(*
SPDX-FileCopyrightText: © 2026 Oleksandr Tiutyk <trofimich@gmail.com>
SPDX-License-Identifier: MIT
License: https://opensource.org/license/mit
*)

(*!
<summary>Defines a boolean predicate evaluated by workflow activities.</summary>
*)

INTERFACE ICondition EXTENDS IWorkflowElement

(*!
<summary>Reports whether the condition is completely configured and ready for evaluation.</summary>
*)
{attribute 'monitoring' := 'call'}
PROPERTY Configured : BOOL
GET
END_GET
END_PROPERTY

(*!
<summary>Evaluates the condition in the context of the specified activity.</summary>
<param name="activity">Activity requesting evaluation, used for variable lookup context.</param>
*)
METHOD Evaluate : BOOL
VAR_INPUT
	activity : IActivity;
END_VAR
END_METHOD

(*!
<summary>Resolves the nearest activity that hosts this condition, traversing parent conditions if needed.</summary>
<description>
Returns the direct ParentActivity when attached directly to an activity, or traverses the ParentCondition
chain upward until the hosting activity is found. Returns 0 if unattached.
</description>
*)
{attribute 'monitoring' := 'call'}
PROPERTY EnclosingActivity : IActivity
GET
END_GET
END_PROPERTY

(*!
<summary>Gets or sets the borrowed immediate parent activity to which this condition is attached.</summary>
<description>
Returns 0 when the condition is attached to a parent condition rather than directly to an activity.
Use EnclosingActivity to resolve the owning activity context through the parent condition chain.
The standard implementation validates cycles, fixed workflow association and PASSIVE_READY before a new
link is stored. Existing parent links cannot be detached or replaced; an unchanged link is a no-op.
Parents are borrowed for the tree lifetime and do not transfer ownership. Configuration is single-task
without reentry; a child with a known owner requires a parent from that same known workflow.
</description>
*)
{attribute 'monitoring' := 'call'}
PROPERTY ParentActivity : IActivity
GET
END_GET
SET
END_SET
END_PROPERTY

(*!
<summary>Gets or sets the borrowed parent composite condition to which this condition is attached.</summary>
<description>
The standard implementation validates cycles, fixed workflow association and PASSIVE_READY before a new
link is stored. Existing parent links cannot be detached or replaced; an unchanged link is a no-op.
Parents are borrowed for the tree lifetime and do not transfer ownership. Configuration is single-task
without reentry; a child with a known owner requires a parent from that same known workflow.
</description>
*)
{attribute 'monitoring' := 'call'}
PROPERTY ParentCondition : ICondition
GET
END_GET
SET
END_SET
END_PROPERTY

END_INTERFACE

(* stored: Version 1.1.0.1
   Itf ICondition: Id {19c0280f-d2f8-424c-8f16-7278f6083af3}
   Property Configured: Id {be75d7d4-64bd-40dc-bf90-f31d9ada671d}
   Get Get: Id {2cba87ee-59ce-4e78-adf7-b7ddc27d2a6b}
   Method Evaluate: Id {10c78263-1c71-45c9-9b13-37be129d2d1c}
   Property EnclosingActivity: Id {bafd7227-41ac-4f1b-8902-4752d6ce1cbf}
   Get Get: Id {36cff938-a908-479f-9391-58af2b4987b2}
   Property ParentActivity: Id {336055e4-538d-4d26-b32a-4579c4dcea29}
   Get Get: Id {ee7ae3cd-f785-417e-8de6-667289c8af2c}
   Set Set: Id {5479ead8-c01c-4380-b506-f2519cf912ad}
   Property ParentCondition: Id {0792b032-8252-41bb-9047-1e6672dce56a}
   Get Get: Id {86296be7-b61a-41e6-9fb5-4e1edf3638e3}
   Set Set: Id {082ef0f0-de40-45ce-9b96-9039bdbdf281} *)
